PROGRAM MAIN
VAR
END_VAR

END_PROGRAM

(* stored: Version 1.1.0.1
   POU MAIN: Id {9d1c8039-000a-46b5-bba2-99bd9f79b70b} *)
